// TwinCAT 3 PLC project IotFunctionsSamples
// ProgramVersion: 3.1.4022.2
// libraries:
//   Tc2_Standard, * (Beckhoff Automation GmbH)
//   Tc2_System, * (Beckhoff Automation GmbH)
//   Tc2_Utilities, * (Beckhoff Automation GmbH)
//   Tc3_IotFunctions, * (Beckhoff Automation GmbH)
//   Tc3_Module, * (Beckhoff Automation GmbH)
// project tree:
//   / PlcTask.TcTTO
//   POUs/ IotFunctionsSampleA.TcPOU, IotFunctionsSampleB.TcPOU, IotFunctionsSampleC.TcPOU
// real-time tasks:
//   TASK PlcTask: cycle T#10ms, priority 20, ADS port 350

CONFIGURATION IotFunctionsSamples
    RESOURCE PLC ON TwinCAT3
        TASK PlcTask(INTERVAL := T#10ms, PRIORITY := 20);
        PROGRAM IotFunctionsSampleB WITH PlcTask : IotFunctionsSampleB;
    END_RESOURCE
END_CONFIGURATION

// ---- POUs/IotFunctionsSampleB.TcPOU
(*
This sample utilizes a request (fbRequest) to synchronize multiple read operations (aRead[0..4])
*)
PROGRAM IotFunctionsSampleB
VAR
	//IotFunctions specific FB declarations
	fbConnector 	: FB_IotFunctions_Connector := (sAmsNetId := '127.0.0.1.1.1',nDefaultRequesttimeout := 3000,nDefaultMessageRetryInterval := 750);
	fbWrite      	: FB_IotFunctions_Message 	:= (nChannelId := 1);
	aRead 			: ARRAY[0..4] OF FB_IotFunctions_Message 	:= 
																	[(nChannelId := 1)
																	,(nChannelId := 1)
																	,(nChannelId := 1)
																	,(nChannelId := 1)
																	,(nChannelId := 1)
																	];
	fbRequest		: FB_IotFunctions_Request := (nRequestTimeout := 10000);
	
	//sample specific variables.
	nOut 							: UDINT;
	aIn  							: ARRAY[0..4] OF UDINT; // aIn
	nIdx							: UDINT;
	
	aCountSuccessRead				: ARRAY[0..4] OF UDINT;
	aCountSuccessReadDataAvailable	: ARRAY[0..4] OF UDINT;
	aCountSuccessReadDataChanged	: ARRAY[0..4] OF UDINT;
	nCountSuccessWrite				: UDINT;
	
	aCountErrorRead 				: ARRAY[0..4] OF UDINT;	
	nCountErrorWrite 				: UDINT;

	nCountErrorRequest 				: UDINT;
	nCountErrorTimeout 				: UDINT;
	bWrite							: BOOL;
	
	bConnectorError					: BOOL;
END_VAR

nOut := nOut + 1;




// Mandatory call to Execute()
fbConnector.Execute(); 

//Optional way to react to ANY error having occurred during Execute.
IF fbConnector.bError THEN
	bConnectorError := TRUE;
END_IF

IF NOT fbRequest.bBusy THEN
	//error handling
	IF fbRequest.bError THEN
		// Will be triggered when at least one of the included message operations throws an error
		nCountErrorRequest := nCountErrorRequest + 1;		
		//Check individual read message error status [shown as a for-loop]
		FOR nIdx := 0 TO 4 BY 1 DO
			IF aRead[nidx].bError THEN
				aCountErrorRead[nidx] := aCountErrorRead[nidx] + 1;
				aRead[nIdx].Acknowledge();
			END_IF
		END_FOR
		//check fbWrite error status.
		IF fbWrite.bError THEN
			nCountErrorWrite := nCountErrorWrite +1;
			fbWrite.Acknowledge();
		END_IF
	END_IF	
	//timeout handling (timeouts will also occur if at least one included message was not able to retrieve data from target channel prior to timeout)  
	IF fbRequest.bTimeoutOccurred THEN
		// Will be triggered when at least one of the included message operations times out (RequestTimeout)
		nCountErrorTimeout := nCountErrorTimeout + 1;
	END_IF
	
	//Check individual read message success status [shown as a for-loop]
	FOR nIdx := 0 TO 4 BY 1 DO
		IF aRead[nIdx].bSuccess THEN
			//general case of success: no error occurred for this message
			aCountSuccessRead[nidx] := aCountSuccessRead[nidx] + 1;
			IF aRead[nIdx].bDataAvailable THEN
				//data was read from the target channel
				aCountSuccessReadDataAvailable[nIdx] := aCountSuccessReadDataAvailable[nIdx] + 1;
			END_IF
			IF aRead[nIdx].bDataChanged THEN
				//data was read from the target channel and differs from previously contained data in associated symbol (in this case: nIn array)
				aCountSuccessReadDataChanged[nIdx] := aCountSuccessReadDataChanged[nIdx] + 1;
			END_IF
		END_IF
	END_FOR
	
	// Start the new request
	fbRequest.Create();
	fbRequest.EnqueueRead(pMessageFB := ADR(aRead[0]), pPayload := ADR(aIn[0]), nPayloadSize := SIZEOF(aIn[0]));		
	fbRequest.EnqueueRead(pMessageFB := ADR(aRead[1]), pPayload := ADR(aIn[1]), nPayloadSize := SIZEOF(aIn[1]));
	fbRequest.EnqueueRead(pMessageFB := ADR(aRead[2]), pPayload := ADR(aIn[2]), nPayloadSize := SIZEOF(aIn[2]));
	fbRequest.EnqueueRead(pMessageFB := ADR(aRead[3]), pPayload := ADR(aIn[3]), nPayloadSize := SIZEOF(aIn[3]));
	fbRequest.EnqueueRead(pMessageFB := ADR(aRead[4]), pPayload := ADR(aIn[4]), nPayloadSize := SIZEOF(aIn[4]));
	fbRequest.Execute();
	
END_IF 

//data source - this can be any external data source that writes to the configured channel
//for the purpose of this sample, setting the bWrite flag of the sample code to true will result in a single write operation to the specified channel.
IF NOT fbwrite.bBusy THEN
	IF fbWrite.bError THEN
		nCountErrorWrite 	:= nCountErrorWrite + 1;
	ELSIF fbWrite.bSuccess THEN
		nCountSuccessWrite 	:= nCountSuccessWrite + 1;
	END_IF
	fbwrite.Acknowledge();
	IF bWrite THEN
		fbwrite.Write(ADR(nOut),SIZEOF(nOut));
		
		bWrite := FALSE;
	END_IF
END_IF

END_PROGRAM

// ---- POUs/IotFunctionsSampleA.TcPOU
(*
This sample utilizes two message FBs to realize a read operation (fbRead) and a write operation (fbWrite).
*)
PROGRAM IotFunctionsSampleA
VAR
	//creates a FB_IotFunctions_Connector for the Data Agent instance running at the specified sAmsNetId. 
	//(if Data Agent and IotFunctions runtime are on the same machine, the default (127.0.0.1.1.1) will suffice.
	fbConnector : FB_IotFunctions_Connector := (sAmsNetId := '127.0.0.1.1.1');
	//creates a FB_IotFunctions_Message FB intended to be used to read from channel with Id 2. This message will use a timeout of 3s and retry interval of 1s.
	fbRead		: FB_IotFunctions_Message := (nChannelId :=1, nMessageRetryInterval := 1000, nRequestTimeout := 3000);	
	//creates a FB_IotFunctions_Message FB intended to be used to write to channel with Id 2. 10s timeout, 1s retry interval. 
	fbWrite		: FB_IotFunctions_Message := (nChannelId :=1, nMessageRetryInterval := 1000, nRequestTimeout := 10000);

	//sample specific declarations.	
	nIn  				: UDINT := 0;
	nOut 				: UDINT := 1;
	nCountReadData 		: UDINT := 0;
	nCountWriteError 	: UDINT := 0;	
	nCountReadError 	: UDINT := 0;
	bWrite 				: BOOL;
	bConnectorError 	: BOOL;
	
END_VAR

nOut := nOut + 1 ;
fbConnector.Execute();

//optional way to react to ANY error having occurred during Execute.
IF fbConnector.bError THEN
	bConnectorError := TRUE;
END_IF

//error handling
IF fbConnector.bError THEN
	IF fbRead.bError THEN
		nCountReadError := nCountReadError + 1;
		fbRead.Acknowledge();
	END_IF
	IF fbWrite.bError THEN
		nCountWriteError := nCountWriteError + 1;
		fbWrite.Acknowledge();
	END_IF
END_IF


IF fbRead.bDataAvailable THEN
	//handle data that has been read from target channel.
	nCountReadData := nCountReadData +1;
END_IF

//start read operation [note that invoking Read implicitly checks if the FB is busy - invoking Read on an ongoing Read operation therefore will not override the ongoig operation!]
//if you want to abort an ongoing operation, you can invoke Reset.
fbRead.Read(ADR(nIn),SIZEOF(nIn));

//data source - this can be any external data source that writes to the configured channel
//for the purpose of this sample, setting the bWrite flag of the sample code to true will result in a single write operation to the specified channel.
IF bWrite THEN
	IF NOT fbWrite.bBusy THEN
		bWrite := FALSE;
		fbWrite.Write(ADR(nOut),SIZEOF(nOut));		
	END_IF
END_IF

END_PROGRAM

// ---- POUs/IotFunctionsSampleC.TcPOU
(*
This sample combines singular message operations (aRead[10], aWrite[1]), synchronized read operations with requests (aRead[0..4] governed by aRequest[1])
and synchronized read and write operation with requests (aRead[5..9] and aWrite[2] governed by aRequest[2]).
*)
PROGRAM IotFunctionsSampleC
VAR
	//IotFunctions specific FB declarations
	fbConnector 	: FB_IotFunctions_Connector := (sAmsNetId := '127.0.0.1.1.1',nDefaultRequesttimeout := 3000,nDefaultMessageRetryInterval := 750);
	
	aWrite			: ARRAY[1..2] OF FB_IotFunctions_Message := [(nChannelId := 1)
																,(nChannelId := 1)
																];


	aRead 			: ARRAY[0..10] OF FB_IotFunctions_Message 	:= 
																	[(nChannelId := 1)
																	,(nChannelId := 1)
																	,(nChannelId := 1)
																	,(nChannelId := 1)
																	,(nChannelId := 1)																	
																	,(nChannelId := 1)
																	,(nChannelId := 1)
																	,(nChannelId := 1)
																	,(nChannelId := 1)
																	,(nChannelId := 1)																	
																	,(nChannelId := 1)
																	];
																	
	aRequest		: ARRAY[1..2] OF FB_IotFunctions_Request := [(nRequestTimeout := 10000)
																,(nRequestTimeout := 15000)
																];																	
																	

	
	//sample specific variables.
	bOnlineChange					: BOOL;
	nOut 							: UDINT;
	aIn  							: ARRAY[0..10] OF UDINT; // aIn
	nIdx							: UDINT;
	
	//status counter for fbRead[0..10] 
	aCountSuccessRead				: ARRAY[0..10] OF UDINT;
	aCountSuccessReadDataAvailable	: ARRAY[0..10] OF UDINT;
	aCountSuccessReadDataChanged	: ARRAY[0..10] OF UDINT;
	aCountErrorRead 				: ARRAY[0..10] OF UDINT;	
	aCountErrorTimeout 				: ARRAY[0..10] OF UDINT;
	
	//status counter for fbWrite
	aCountSuccessWrite				: ARRAY[1..2] OF UDINT;
	aCountErrorWrite 				: ARRAY[1..2] OF UDINT;
	
	
	//status counter for requests
	aCountErrorRequest 				: ARRAY[1..2] OF UDINT;
	
	bWrite							: BOOL;
	bConnectorError					: BOOL;
	
	bReset							: BOOL;
	
END_VAR

nOut := nOut + 1;

//Mandatory call to Execute()
fbConnector.Execute(); 

//Optional way to react to ANY error having occurred during Execute.
IF fbConnector.bError THEN
	bConnectorError := TRUE;
END_IF

//Using the aRead[10] FB to realize a standalone read operation.
IF NOT aRead[10].bBusy THEN
	IF aRead[10].bError THEN
		aCountErrorRead[10] := aCountErrorRead[10] +1 ;
	END_IF	
	IF aRead[10].bTimeoutOccurred THEN
		aCountErrorTimeout[10] := aCountErrorTimeout[10] +1 ;
	END_IF	
	IF aRead[10].bSuccess THEN
		//general case of success: no error occurred for this message
		aCountSuccessRead[10] := aCountSuccessRead[10] + 1;
		IF aRead[10].bDataAvailable THEN
			//data was read from the target channel
			aCountSuccessReadDataAvailable[10] := aCountSuccessReadDataAvailable[10] + 1;
		END_IF
		IF aRead[10].bDataChanged THEN
			//data was read from the target channel and differs from previously contained data in associated symbol (in this case: nIn array)
			aCountSuccessReadDataChanged[10] := aCountSuccessReadDataChanged[10] + 1;
		END_IF
	END_IF
	
	//Start new read operation.
	aRead[10].Read(pPayload := ADR(aIN[10]),nPayloadSize := SIZEOF(aIn[10]));
END_IF

// aRequest[1] governing aRead[0..4]
IF NOT aRequest[1].bBusy THEN

	IF aRequest[1].bError THEN
		// Will be triggered when at least one of the included message operations throws an error
		aCountErrorRequest[1] := aCountErrorRequest[1] + 1;			
		//Check individual read message error status [shown as a for-loop]
		FOR nIdx := 0 TO 4 BY 1 DO
			IF aRead[nIdx].bError THEN
				aCountErrorRead[nIdx] := aCountErrorRead[nIdx] + 1;
				aRead[nIdx].Acknowledge();
			END_IF
		END_FOR

	END_IF	
	//timeout handling (timeouts will also occur if at least one included message was not able to retrieve data from target channel prior to timeout)  
	IF aRequest[1].bTimeoutOccurred THEN
		// Will be triggered when at least one of the included message operations times out (RequestTimeout)
		
		FOR nIdx := 0 TO 4 BY 1 DO
			IF aRead[nIdx].bTimeoutOccurred THEN
				//this message has timed out.
				aCountErrorTimeout[nIdx] := aCountErrorTimeout[nIdx] + 1;
			END_IF
		END_FOR
	END_IF
	
	//Check individual read message success status [shown as a for-loop]
	FOR nIdx := 0 TO 4 BY 1 DO
		IF aRead[nIdx].bSuccess THEN
			//general case of success: no error occurred for this message
			aCountSuccessRead[nidx] := aCountSuccessRead[nidx] + 1;
			IF aRead[nIdx].bDataAvailable THEN
				//data was read from the target channel
				aCountSuccessReadDataAvailable[nIdx] := aCountSuccessReadDataAvailable[nIdx] + 1;
			END_IF
			IF aRead[nIdx].bDataChanged THEN
				//data was read from the target channel and differs from previously contained data in associated symbol (in this case: nIn array)
				aCountSuccessReadDataChanged[nIdx] := aCountSuccessReadDataChanged[nIdx] + 1;
			END_IF
		END_IF
	END_FOR
	
	// Start the new request
	aRequest[1].Create();
	aRequest[1].EnqueueRead(pMessageFB := ADR(aRead[0]), pPayload := ADR(aIn[0]), nPayloadSize := SIZEOF(aIn[0]));		
	aRequest[1].EnqueueRead(pMessageFB := ADR(aRead[1]), pPayload := ADR(aIn[1]), nPayloadSize := SIZEOF(aIn[1]));
	aRequest[1].EnqueueRead(pMessageFB := ADR(aRead[2]), pPayload := ADR(aIn[2]), nPayloadSize := SIZEOF(aIn[2]));
	aRequest[1].EnqueueRead(pMessageFB := ADR(aRead[3]), pPayload := ADR(aIn[3]), nPayloadSize := SIZEOF(aIn[3]));
	aRequest[1].EnqueueRead(pMessageFB := ADR(aRead[4]), pPayload := ADR(aIn[4]), nPayloadSize := SIZEOF(aIn[4]));
	aRequest[1].Execute();
	
END_IF 

// aRequest[2] governing aRead[5..9]
IF NOT aRequest[2].bBusy THEN
	IF aRequest[2].bError THEN
		// Will be triggered when at least one of the included message operations throws an error
		aCountErrorRequest[2] := aCountErrorRequest[2] + 1;		
		//Check individual read message error status [shown as a for-loop]
		FOR nIdx := 5 TO 9 BY 1 DO
			IF aRead[nIdx].bError THEN
				aCountErrorRead[nIdx] := aCountErrorRead[nIdx] + 1;
				aRead[nIdx].Acknowledge();
			END_IF
		END_FOR
		IF aWrite[2].bError THEN
			aCountErrorWrite[2] := aCountErrorWrite[2] +1;
			aWrite[2].Acknowledge();
		END_IF
	END_IF	
	
	//Timeout handling (timeouts will also occur if at least one included message was not able to retrieve data from target channel prior to timeout)  
	IF aRequest[2].bTimeoutOccurred THEN
		// Will be triggered when at least one of the included message operations times out (RequestTimeout)
		FOR nIdx := 5 TO 9 BY 1 DO
			IF aRead[nIdx].bTimeoutOccurred THEN
				//this message has timed out.
				aCountErrorTimeout[nIdx] := aCountErrorTimeout[nIdx] + 1;
			END_IF
		END_FOR
	END_IF
	
	//Check individual read message success status [shown as a for-loop]
	FOR nIdx := 5 TO 9 BY 1 DO
		IF aRead[nIdx].bSuccess THEN
			//general case of success: no error occurred for this message
			aCountSuccessRead[nidx] := aCountSuccessRead[nidx] + 1;
			IF aRead[nIdx].bDataAvailable THEN
				//data was read from the target channel
				aCountSuccessReadDataAvailable[nIdx] := aCountSuccessReadDataAvailable[nIdx] + 1;
			END_IF
			IF aRead[nIdx].bDataChanged THEN
				//data was read from the target channel and differs from previously contained data in associated symbol (in this case: nIn array)
				aCountSuccessReadDataChanged[nIdx] := aCountSuccessReadDataChanged[nIdx] + 1;
			END_IF
		END_IF
	END_FOR
	IF aWrite[2].bSuccess THEN
		aCountSuccessWrite[2] 	:= aCountSuccessWrite[2] + 1;
	END_IF
	
		// Start the new request
	aRequest[2].Create();
	aRequest[2].EnqueueRead(pMessageFB := ADR(aRead[5]), pPayload := ADR(aIn[5]), nPayloadSize := SIZEOF(aIn[5]));		
	aRequest[2].EnqueueRead(pMessageFB := ADR(aRead[6]), pPayload := ADR(aIn[6]), nPayloadSize := SIZEOF(aIn[6]));
	aRequest[2].EnqueueRead(pMessageFB := ADR(aRead[7]), pPayload := ADR(aIn[7]), nPayloadSize := SIZEOF(aIn[7]));
	aRequest[2].EnqueueRead(pMessageFB := ADR(aRead[8]), pPayload := ADR(aIn[8]), nPayloadSize := SIZEOF(aIn[8]));
	aRequest[2].EnqueueRead(pMessageFB := ADR(aRead[9]), pPayload := ADR(aIn[9]), nPayloadSize := SIZEOF(aIn[9]));
	aRequest[2].EnqueueWrite(pMessageFB := ADR(aWrite[2]), pPayload := ADR(nOut), nPayloadSize := SIZEOF(nOut));
	aRequest[2].Execute();
	
END_IF

//data source - this can be any external data source that writes to the configured channel
//for the purpose of this sample, setting the bWrite flag of the sample code to true will result in a single write operation to the specified channel.

// attempt to start a write operation every 100th cycle.
IF nOut MOD 100 = 0 THEN
	bWrite := true;
END_IF

IF NOT aWrite[1].bBusy THEN
	IF aWrite[1].bError THEN
		aCountErrorWrite[1] := aCountErrorWrite[1] + 1;
		aWrite[1].Acknowledge();
	ELSIF aWrite[1].bSuccess THEN
		aCountSuccessWrite[1] := aCountSuccessWrite[1] + 1;
		aWrite[1].Acknowledge();
	END_IF
	IF bWrite THEN
		aWrite[1].Write(ADR(nOut),SIZEOF(nOut));
		bWrite := FALSE;	
	END_IF
END_IF

END_PROGRAM
